{attribute addProperty BoxType "EL1258-0000-0016"}
{attribute addProperty Id "No_of_input_eventsUSINT811Input_stateBIT10.1259Input_buffer_overflowBIT10.12510Input_cycle_counter_BIT_0BIT10.12515Input_cycle_counter_BIT_1BIT10.12515Events_in_input_bufferUSINT8117Input_order_feedbackUSINT8118"}
{attribute addProperty CRC "2239177261"}
{attribute addProperty SizeInBites "60"}
{attribute addProperty SizeInBytes "7.5"}
{warning 'Size of this structure is not a multiple of 8 bits!!!'}
TYPE Status_8577222D :
STRUCT
	{attribute addProperty Name "No_of_input_events"}
	No_of_input_events : USINT;
	{attribute addProperty Name "Input_state"}
	Input_state : BIT;
	{attribute addProperty Name "Input_buffer_overflow"}
	Input_buffer_overflow : BIT;
	{attribute 'hide'}
	reserve_1_BOOL_0 : BOOL;
	{attribute 'hide'}
	reserve_1_BOOL_1 : BOOL;
	{attribute 'hide'}
	reserve_1_BOOL_2 : BOOL;
	{attribute 'hide'}
	reserve_1_BOOL_3 : BOOL;
	{attribute addProperty Name "Input_cycle_counter"}
	Input_cycle_counter_BIT_0 : BIT;
	{attribute addProperty Name "Input_cycle_counter"}
	Input_cycle_counter_BIT_1 : BIT;
	{attribute addProperty Name "Events_in_input_buffer"}
	Events_in_input_buffer : USINT;
	{attribute addProperty Name "Input_order_feedback"}
	Input_order_feedback : USINT;
END_STRUCT
END_TYPE

(* stored: Version 1.2.0.0, ProductVersion 3.1.4024.9
   DUT Status_8577222D: Id {60e661f5-c19d-4d81-afcd-cd5b3c40a7e6} *)
